(* PLC project  *)

PROGRAM hugo

END_PROGRAM

PROGRAM bert/bart

END_PROGRAM

PROGRAM dupli

END_PROGRAM

PROGRAM dupli

END_PROGRAM

CONFIGURATION Device
END_CONFIGURATION

CONFIGURATION Foo
END_CONFIGURATION
